// TIA Portal V16 export
// export: Created 2022-08-03T14:37:59.2955471Z, ExportSetting WithDefaults, DisplayName Totally Integrated Automation Portal, DisplayVersion V16, DisplayName TIA Portal Version Control Interface, DisplayVersion V16, DisplayName TIA Portal Openness, DisplayVersion V16, DisplayName SINAMICS Startdrive Advanced, DisplayVersion V16, DisplayName SINAMICS Startdrive G130, G150, S120, S150, SINAMICS MV, S210, DisplayVersion V16, DisplayName SINAMICS Startdrive G110M, G120, G120C, G120D, G120P, DisplayVersion V16, DisplayName STEP 7 Professional, DisplayVersion V16, DisplayName STEP 7 Safety, DisplayVersion V16, DisplayName WinCC Professional, DisplayVersion V16
VAR_GLOBAL   // PLC tag table "Electrical_interlock tag table"
   Stop AT %I0.0 : Bool;
   Start AT %I0.1 : Bool;
   Sistem AT %Q0.0 : Bool;
   btn_ileri AT %I0.2 : Bool;
   m_ileri AT %Q0.1 : Bool;
   btn_geri AT %I0.3 : Bool;
   m_geri AT %Q0.2 : Bool;
END_VAR
